Staubli VAL3: setConvSpeed.pgx

program setConvSpeed(num x_nConvNum (dimensions=1), num& x_nError[] (dimensions=1))
begin
  // This program updates the speed of the conveyor on the conveyor library
  //
  // Input Param
  //  x_nConvNum  : Conveyor number
  //
  // Output Param
  //  x_nError    : Error code
  //    0    --> No error
  //    3    --> Invalid conveyor number
  //
  //----------------------------------------------------------------
  //
  x_nError=0
  switch x_nConvNum
    case 0
      cnv0:nConveyorSpeed=nConveyorSpeed[x_nConvNum]
    break
    case 1
      cnv1:nConveyorSpeed=nConveyorSpeed[x_nConvNum]
    break
    default
      x_nError=3
    break
  endSwitch
end
